Omron Sysmac Studio project 210907_PLC_FINS_Python_control (Sysmac Studio 1.45.1.64010, StandardProject)

# Controller new_Controller_0: NJ301-1100 version 1.9
Units and slaves: 전원 : NJ-Px3001; CPU : NJ301-1100; 0 : CJ1W-ID231 (J01); 1 : CJ1W-OD231 (J02)
Axis Node2, settings changed from default: AxisType=ServoType, UnitsConversion=EnumElement2, UnitsNumerator=1048576, UnitsDenominator=90, MaxVelocity=4500, MaxJogVelocity=4500, InPositionBand=0.1, ZeroPositionBand=0.1, CountMode=EnumElement2, ModuloMAXPosition=400, ModuloMINPosition=0
Axis Node3, settings changed from default: AxisNumber=1, AxisType=ServoType, UnitsConversion=EnumElement5, UnitsNumerator=131072, UnitsDenominator=360, MaxVelocity=18000, MaxJogVelocity=18000, InPositionBand=0.1, ZeroPositionBand=0.1, CountMode=EnumElement2, ModuloMAXPosition=400, ModuloMINPosition=0
Axes group MC_Group000, settings changed from default: GroupGroupUse=GroupUsingGroup, GroupMaxVelocity=10000
Task PrimaryTask (priority 4, period or condition 2000): Program0

VAR_GLOBAL RETAIN
    GD AT %D0 : ARRAY[0..99] OF BYTE;
END_VAR
VAR_GLOBAL
    GM AT %0 : ARRAY[0..99] OF BOOL;
    Name : STRING[256];  (* published *)
    EmpolyNumber : STRING[256];  (* published *)
    PhoneNumber : STRING[256];  (* published *)
    ClientRqst : STRING[256];
END_VAR
VAR_GLOBAL CONSTANT
    Node2 : _sAXIS_REF;  (* at MC://_MC_AX[0] *)
    Node3 : _sAXIS_REF;  (* at MC://_MC_AX[1] *)
END_VAR
VAR_GLOBAL
    cyl10 : BOOL;  (* 공급실린더 후진; at IOBus://rack#0/slot#0/Ch1_In/Ch1_In00 *)
    cyl11 : BOOL;  (* 공급실린더 전진; at IOBus://rack#0/slot#0/Ch1_In/Ch1_In01 *)
    cyl20 : BOOL;  (* 흡착실린더 후진; at IOBus://rack#0/slot#0/Ch1_In/Ch1_In02 *)
    cyl21 : BOOL;  (* 흡착실린더 전진; at IOBus://rack#0/slot#0/Ch1_In/Ch1_In03 *)
    cyl30 : BOOL;  (* 이송실린더 후진; at IOBus://rack#0/slot#0/Ch1_In/Ch1_In04 *)
    cyl31 : BOOL;  (* 이송실린더 전진; at IOBus://rack#0/slot#0/Ch1_In/Ch1_In05 *)
    cyl40 : BOOL;  (* 차단실린더 후진; at IOBus://rack#0/slot#0/Ch1_In/Ch1_In06 *)
    cyl41 : BOOL;  (* 차단실린더 전진; at IOBus://rack#0/slot#0/Ch1_In/Ch1_In07 *)
    air1 : BOOL;  (* 진공 흡착 확인; at IOBus://rack#0/slot#0/Ch1_In/Ch1_In08 *)
    lim1 : BOOL;  (* 트레이 리밋스위치 (좌); at IOBus://rack#0/slot#0/Ch1_In/Ch1_In09 *)
    lim2 : BOOL;  (* 트레이 리밋스위치 (우); at IOBus://rack#0/slot#0/Ch1_In/Ch1_In10 *)
    sen3 : BOOL;  (* 용량 센서; at IOBus://rack#0/slot#0/Ch1_In/Ch1_In11 *)
    sen2 : BOOL;  (* 근접 센서; at IOBus://rack#0/slot#0/Ch1_In/Ch1_In12 *)
    sen1 : BOOL;  (* 공급 센서; at IOBus://rack#0/slot#0/Ch1_In/Ch1_In13 *)
    sen4 : BOOL;  (* 차단 센서; at IOBus://rack#0/slot#0/Ch1_In/Ch1_In14 *)
    pos1 : BOOL;  (* 말굽 센서 (우); at IOBus://rack#0/slot#0/Ch1_In/Ch1_In15 *)
    pos2 : BOOL;  (* 말굽 센서 (중); at IOBus://rack#0/slot#0/Ch2_In/Ch2_In00 *)
    pos3 : BOOL;  (* 말굽 센서 (좌); at IOBus://rack#0/slot#0/Ch2_In/Ch2_In01 *)
    pos4 : BOOL;  (* 말굽 센서 (트레이 모터); at IOBus://rack#0/slot#0/Ch2_In/Ch2_In02 *)
    pb1 : BOOL;  (* 스위치 (적); at IOBus://rack#0/slot#0/Ch2_In/Ch2_In03 *)
    pb2 : BOOL;  (* 스위치 (청); at IOBus://rack#0/slot#0/Ch2_In/Ch2_In04 *)
    pb3 : BOOL;  (* 스위치 (토글); at IOBus://rack#0/slot#0/Ch2_In/Ch2_In05 *)
    l1 : BOOL;  (* 램프(황); at IOBus://rack#0/slot#1/Ch1_Out/Ch1_Out00 *)
    l2 : BOOL;  (* 램프(청); at IOBus://rack#0/slot#1/Ch1_Out/Ch1_Out01 *)
    l3 : BOOL;  (* 램프(적); at IOBus://rack#0/slot#1/Ch1_Out/Ch1_Out02 *)
    cyl1 : BOOL;  (* SOL1 공급실린더; at IOBus://rack#0/slot#1/Ch1_Out/Ch1_Out03 *)
    cyl2 : BOOL;  (* SOL2 흡착실린더; at IOBus://rack#0/slot#1/Ch1_Out/Ch1_Out04 *)
    cyl3A : BOOL;  (* SOL3 이송실린더 전진; at IOBus://rack#0/slot#1/Ch1_Out/Ch1_Out05 *)
    cyl3B : BOOL;  (* SOL4 이송실린더 후진; at IOBus://rack#0/slot#1/Ch1_Out/Ch1_Out06 *)
    cyl4 : BOOL;  (* SOL5 차단실린더; at IOBus://rack#0/slot#1/Ch1_Out/Ch1_Out07 *)
    air0 : BOOL;  (* SOL6 진공흡착; at IOBus://rack#0/slot#1/Ch1_Out/Ch1_Out08 *)
    conN : BOOL;  (* 컨베이어 모터 정회전; at IOBus://rack#0/slot#1/Ch1_Out/Ch1_Out09 *)
    traN : BOOL;  (* 트레이 모터 정회전; at IOBus://rack#0/slot#1/Ch1_Out/Ch1_Out10 *)
    traR : BOOL;  (* 트레이 모터 역회전; at IOBus://rack#0/slot#1/Ch1_Out/Ch1_Out11 *)
    conR : BOOL;  (* 컨베이어 모터 역회전; at IOBus://rack#0/slot#1/Ch1_Out/Ch1_Out12 *)
END_VAR
VAR_GLOBAL
    CamProfile0 : ARRAY[0..15000] OF _sMC_CAM_REF := None;
END_VAR

PROGRAM Program0
VAR
    lp1 : BOOL;
    Open : BOOL;
    Socket_1 : _sSOCKET;
    Open1 : SktTCPAccept;
    Rcv1 : SktTCPRcv;
    TcpStatus : _eCONNECTION_STATE;
    DatRcvFlag : BOOL;
    STauts_1 : SktGetTCPStatus;
    BufferC1 : SktClearBuf;
    Close_1 : BOOL;
    RcvD : ARRAY[0..49] OF BYTE;
    ErrorRcv : BOOL;
    snd1 : SktTCPSend;
    Close_2 : BOOL;
    SendD : ARRAY[0..14] OF BYTE;
    ErrorSnd : BOOL;
    SendDD : ARRAY[0..14] OF BYTE;
    SendDDD : ARRAY[0..14] OF BYTE;
    snd2 : SktTCPSend;
    snd3 : SktTCPSend;
    Close1 : SktClose;
    done_opc : BOOL;
    ErrorID1 : WORD;
    ErrorID2 : WORD;
    ErrorID3 : WORD;
    이상해제기동 AT %w0.01 : BOOL;
    EC이상해제 : ResetECError;
    EC이상해제완료 : BOOL;
    EC이상 : BOOL;
    MC이상해제 : ResetMCError;
    컨베이어이상해제기동 AT %w0.02 : BOOL;
    컨베이어이상해제 : MC_Reset;
    원판이상해제기동 AT %w0.03 : BOOL;
    원판이상해제 : MC_Reset;
    서보ON AT %w0.04 : BOOL;
    서보ON유효 : BOOL;
    서보ON중 : BOOL;
    컨베이어ON : MC_Power;
    원판ON : MC_Power;
    서보OFF AT %w0.05 : BOOL;
    녹색램프 AT %w1.01 : BOOL;
    적색램프 AT %w1.02 : BOOL;
    컨에비어조그 AT %w5.10 : BOOL;
    원판조그 AT %w5.11 : BOOL;
    컨베이어조그이송 : MC_MoveJog;
    원판조그이송 : MC_MoveJog;
    data1 : REAL;
    data2 : REAL;
    data3 : REAL;
    data4 : REAL;
    원판원점 : MC_Home;
    컨베이어원점 : MC_Home;
    cam1 : MC_CamIn;
    주축동작 : MC_MoveVelocity;
    Run : BOOL;
    camout1 : MC_CamOut;
    주축정지 : MC_Stop;
END_VAR
VAR_EXTERNAL
    Name : STRING[256];
    EmpolyNumber : STRING[256];
    PhoneNumber : STRING[256];
    ClientRqst : STRING[256];
END_VAR
VAR_EXTERNAL CONSTANT
    Node2 : _sAXIS_REF;
    Node3 : _sAXIS_REF;
END_VAR
VAR_EXTERNAL
    pb3 : BOOL;
    GD : ARRAY[0..99] OF BYTE;
    CamProfile0 : ARRAY[0..15000] OF _sMC_CAM_REF;
    pb1 : BOOL;
    pb2 : BOOL;
END_VAR
VAR
    _e1 : R_TRIG;
    _e2 : R_TRIG;
    _e3 : R_TRIG;
    _e4 : R_TRIG;
    _e5 : R_TRIG;
END_VAR

(* Section Section0: ladder, written here as Structured Text *)

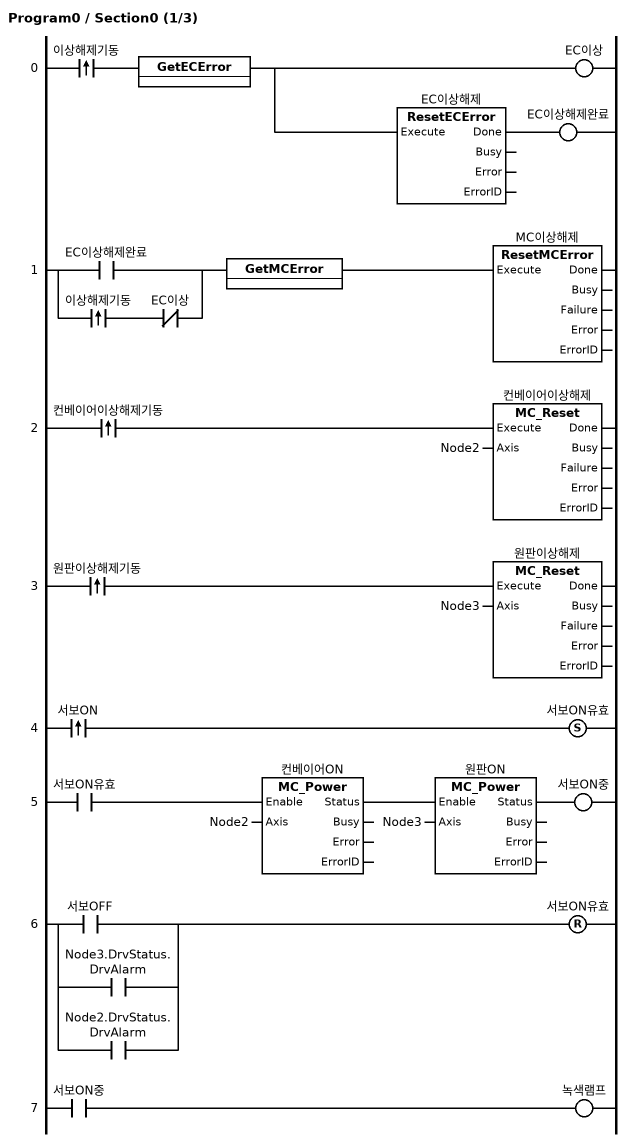
(* Rung 0 *)
_e1(CLK := 이상해제기동);
EC이상 := _e1.Q AND GetECError();
EC이상해제(Execute := _e1.Q AND GetECError());
EC이상해제완료 := EC이상해제.Done;
(* Rung 1 *)
_e2(CLK := 이상해제기동);
MC이상해제(Execute := (EC이상해제완료 OR (_e2.Q AND NOT EC이상)) AND GetMCError());
(* Rung 2 *)
_e3(CLK := 컨베이어이상해제기동);
컨베이어이상해제(Execute := _e3.Q, Axis := Node2);
(* Rung 3 *)
_e4(CLK := 원판이상해제기동);
원판이상해제(Execute := _e4.Q, Axis := Node3);
(* Rung 4 *)
_e5(CLK := 서보ON);
IF _e5.Q THEN 서보ON유효 := TRUE; END_IF;
(* Rung 5 *)
컨베이어ON(Enable := 서보ON유효, Axis := Node2);
원판ON(Enable := 컨베이어ON.Status, Axis := Node3);
서보ON중 := 원판ON.Status;
(* Rung 6 *)
IF 서보OFF OR Node3.DrvStatus.DrvAlarm OR Node2.DrvStatus.DrvAlarm THEN 서보ON유효 := FALSE; END_IF;
(* Rung 7 *)
녹색램프 := 서보ON중;

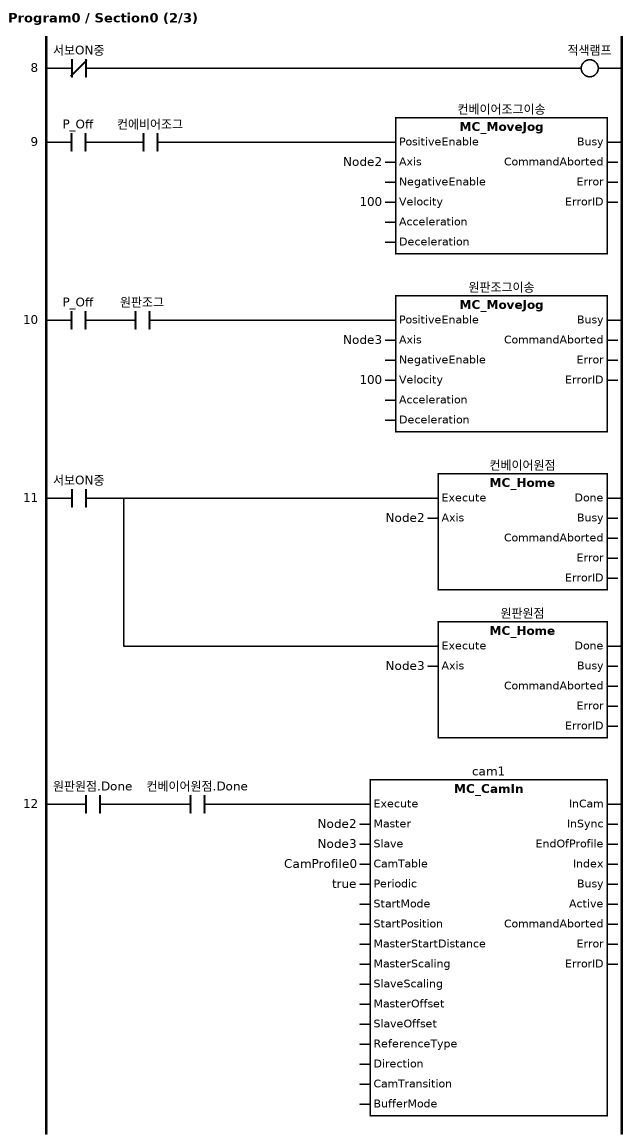
(* Rung 8 *)
적색램프 := NOT 서보ON중;
(* Rung 9 *)
컨베이어조그이송(PositiveEnable := P_Off AND 컨에비어조그, Axis := Node2, Velocity := 100);
(* Rung 10 *)
원판조그이송(PositiveEnable := P_Off AND 원판조그, Axis := Node3, Velocity := 100);
(* Rung 11 *)
컨베이어원점(Execute := 서보ON중, Axis := Node2);
원판원점(Execute := 서보ON중, Axis := Node3);
(* Rung 12 *)
cam1(Execute := 원판원점.Done AND 컨베이어원점.Done, Master := Node2, Slave := Node3, CamTable := CamProfile0, Periodic := true);

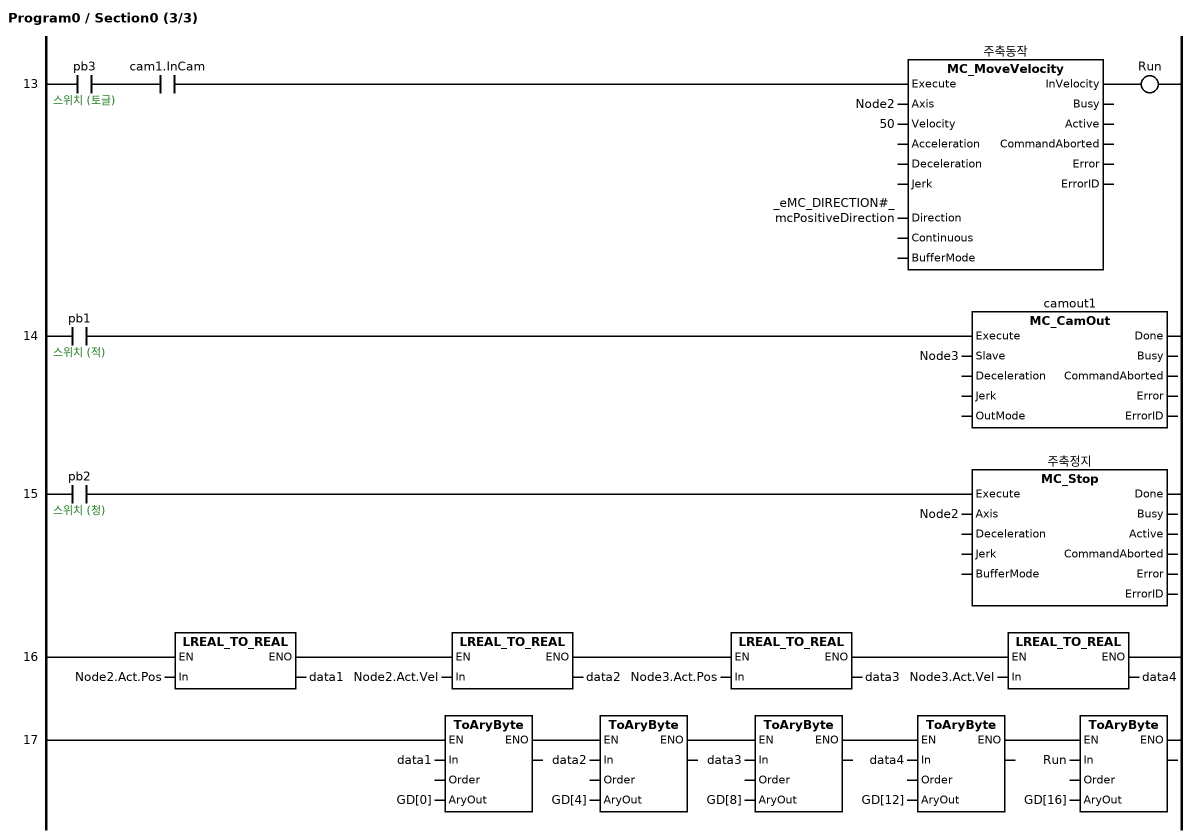
(* Rung 13 *)
주축동작(Execute := pb3 AND cam1.InCam, Axis := Node2, Velocity := 50, Direction := _eMC_DIRECTION#_mcPositiveDirection);
Run := 주축동작.InVelocity;
(* Rung 14 *)
camout1(Execute := pb1, Slave := Node3);
(* Rung 15 *)
주축정지(Execute := pb2, Axis := Node2);
(* Rung 16 *)
data1 := LREAL_TO_REAL(In := Node2.Act.Pos);
data2 := LREAL_TO_REAL(In := Node2.Act.Vel);
data3 := LREAL_TO_REAL(In := Node3.Act.Pos);
data4 := LREAL_TO_REAL(In := Node3.Act.Vel);
(* Rung 17 *)
ToAryByte(In := data1, AryOut := GD[0]);
ToAryByte(In := data2, AryOut := GD[4]);
ToAryByte(In := data3, AryOut := GD[8]);
ToAryByte(In := data4, AryOut := GD[12]);
ToAryByte(In := Run, AryOut := GD[16]);
END_PROGRAM